# EPICS IOC start-up script: examples/test/PSI/epp2038.iocsh
#- mXsXXX naming
require ecmccfg, "NAMING=mXsXXX"

#- add slaves
${SCRIPTEXEC} ${ecmccfg_DIR}addSlave.cmd, "HW_DESC=EPP2038, SLAVE_ID=2"
